(* Logix 5000 project; controller TestController vendor 1 type 14 code 166 rev 32.11; software revision 32.02 *)
// This is a test project

TASK Continuous (continuous, watchdog 500 ms) : MainProgram   // Test continuous task
TASK Event (event, rate 11 ms, priority 10, watchdog 500 ms) : EventProgram   // TestEvent Task
TASK Periodic (periodic, rate 10 ms, priority 10, watchdog 500 ms) : EPProgram, NProgram, Empty

MODULES
   Local : vendor 1 type 14 code 166 (ICP 0, rev 32.11)
      Local_Mod_4 : 1756sc-CTR8 (ICP 4, rev 1.1, Output RPI 10 ms)
      Local_Mod_6 : 1756-CNB (ICP 6, rev 11.1)
         LM6C1 : 1407-CGCM (ControlNet 2, rev 4.1, Output RPI 5 ms)
      Local_Mod_8 : vendor 1 type 14 code 166 (ICP 8, rev 32.1, $6765098e$ RPI 20 ms)
      NetworkController : vendor 1 type 14 code 166 (Ethernet 192.168.1.232, rev 32.1)
      Local_Mod_5 : 1756-M02AE (ICP 5, rev 32.1, MotionEvent RPI 1000 ms, MotionAsync RPI 25 ms)
      TestEtap : 1783-ETAP (Ethernet 192.168.1.247, rev 2.1)
      Local_Mod_1 : 1756-EN2T (ICP 1, Ethernet 1.1.1.1, rev 11.1)
         L1M1 : 1756-EN2T (Ethernet 2.2.2.2, rev 11.1, Output RPI 10 ms)
            L1M1D1 : 1756-IT6I (ICP 1, rev 1.1, Input RPI 100 ms)
         L1M3 : 1732E-IB16M12DR (Ethernet 54.3.56.6, rev 1.1, Input RPI 20 ms)
         L1M2 : 1734-AENT (Ethernet 3.3.3.3, rev 5.1, Output RPI 20 ms)
            L1M2D1 : 1734-IV8 (PointIO 1, rev 3.1)
      RackIO : 1756-EN2T (Ethernet 10.10.10.10, rev 11.1, Output RPI 10 ms)   // This is a test EN2T module
         Rack_Mod_1 : 1756-IB16 (ICP 1, rev 3.1)
         Rack_Mode_3 : 1756-IB16 (ICP 3, rev 3.1)
              RackIO:3:I.Data.0   // IO Description
         Rack_Mod_2 : 1756-IF8 (ICP 2, rev 1.1, Input RPI 100 ms)   // Ths is a test IF8
      TestCard : 1756-EN2T (Ethernet Host-Name.Com1234d5asdvdlkjadvasdfasdfasddfasdfasdfasdasdfasdfda, rev 11.1)   // This is a test EN2T module
      ImportTest : 1756-EN2T (ICP 7, Ethernet 10.2.10.4, rev 11.1)   // This is a test EN2T module
      FlexBus : 1794-AENT (Ethernet 192.168.1.251, rev 4.1, Output RPI 20 ms)
         FB1 : 1794-IB16 (Flex 0, rev 1.1)
         FB2 : 1794-IB16 (Flex 1, rev 1.1)
      Local_Mod_9 : 1756-DHRIO (ICP 9, rev 7.1, Input RPI 25 ms)
         RIOChA1 : 1747-ASB (RIO 1, rev 1.1, Output RPI 48 ms)
         RIOChA2 : 1794-ASB (RIO 2, rev 1.1, Output RPI 48 ms)
         RIOChB1 : 1771-ASB (RIO 0, rev 1.1, Output RPI 48 ms)
      Local_Mod_3 : 1756-RIO (ICP 3, rev 3.1, Output RPI 20 ms)
      Local_Mod_2 : MVI56E-MCM (ICP 2, rev 3.1, Output RPI 5 ms)
      FlexIO : 5094-AEN2TR (Ethernet 10.11.12.13, rev 4.1)
         Flex_Mod_1 : 5094-IF8 (5094 1, rev 2.1, StandardDataDriven RPI 100 ms)
         Flex_Mod_2 : 5094-OB16 (5094 2, rev 2.1, StandardDataDriven RPI 5 ms)
         Flex_Mod_3 : 5094-IB16 (5094 3, rev 2.1, StandardDataDriven RPI 5 ms)
         Flex_Mod_4 : 5094-IB32 (5094 4, rev 2.1, StandardDataDriven RPI 5 ms)
         Flex_Mod_5 : 5094-OF8 (5094 5, rev 2.1, StandardDataDriven RPI 100 ms)
         Flex_Mod_6 : 5094-IY8 (5094 6, rev 3.1, StandardDataDriven RPI 100 ms)
         Flex_Mod_7 : 5094-HSC (5094 7, rev 2.1, StandardDataDriven RPI 80 ms)
END_MODULES

TYPE AlarmType :   // This is a test alarm type
STRUCT
   DigitalMember : CAM;   // Test digital member
END_STRUCT
END_TYPE

TYPE BoolTest :   // This is a test
STRUCT
   Member01 : BOOL;
   Member02 : BOOL;
   Member04 : BOOL;
   Member05 : BOOL;
END_STRUCT
END_TYPE

TYPE FakeString :   // This is a type
STRUCT
   LEN : DINT;
   DATA : SINT[23];
END_STRUCT
END_TYPE

TYPE ModuleType :   // This is a test of a type that references Module-Defined types
STRUCT
   AIChannel : CHANNEL_AI:O:0;   // This is a test
   TestChannel : CHANNEL_AI:O:0;   // This is a test
END_STRUCT
END_TYPE

TYPE MyStringType :   // This is a test string type
STRUCT
   LEN : DINT;
   DATA : SINT[100];
END_STRUCT
END_TYPE

TYPE TestType :   // this is a test
STRUCT
   Timers : TIMER[5];
   Number : DINT;
   Flag : BOOL;
END_STRUCT
END_TYPE

ADD_ON_INSTRUCTION aoi_Test   (* revision 1.2 *)
// Help:
// This is a test aoi definitio that was built for purposes of exporting data to examine the structure of the L5X
VAR_INPUT
   InputTest : BOOL; {visible}
   OutputTest : DINT; {access Read Only, visible}
END_VAR
VAR_IN_OUT
   InOutTest : SimpleType; {required}
END_VAR
VAR_INPUT
   Config : INT; {access None, required}
   Test : BOOL; {access None}
END_VAR
VAR_IN_OUT
   InOutArray : REAL[5]; {required}
END_VAR
VAR_INPUT
   New : DINT; {required}
   Alias : ALIAS FOR LocalBool; {access None}   // This is an alias
END_VAR
VAR
   LocalBool : BOOL; {access None}
   LocalComplex : SimpleType;   // Description Test
   LocalArray : DINT[5]; {access None}
   LocalString : STRING; {access None}
END_VAR

ROUTINE Logic   (* ladder *)
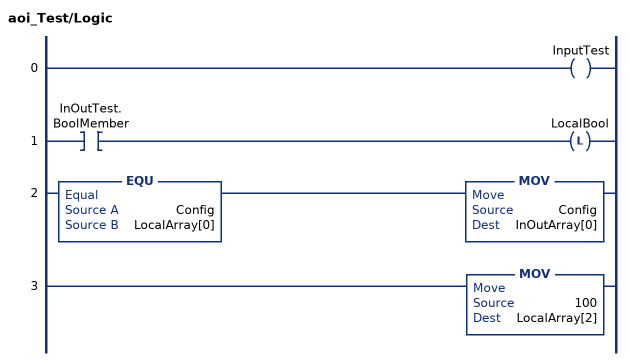
   0: OTE(InputTest);
   1: XIC(InOutTest.BoolMember)OTL(LocalBool);
   2: EQU(Config,LocalArray[0])MOV(Config,InOutArray[0]);
   3: MOV(100,LocalArray[2]);
END_ROUTINE

ROUTINE Prescan   (* ladder *)
END_ROUTINE
END_ADD_ON_INSTRUCTION

VAR_GLOBAL   (* controller tags *)
   _Test : DINT;
   AliasTag : ALIAS FOR Another;
   Another : DINT := 4;
   aoiTestInstance : aoi_Test;
   AsciiTag : SINT := '$10';
   Consumer : DINT;
   DateTimeNs : LINT := 1641016800100100100;
   EPProgram : PHASE;
   FakeStringTag : FakeString;
   MultiDimensionalArray : DINT[3,5];
   NewTag : ComplexType; {access None}
   ProducedTag : DINT; {produced}
   ProviderTag : TIMER; {produced}
   RealArray : REAL[5];
   SimpleArray : DINT[10]; {access Read Only}   // This is a test
   SimpleBool : BOOL;   // A simple boolean tag element
   SimpleDint : DINT := 123392; {access None}
   SimpleInt : INT := 4321; {access None}   // This is a simple integer tag
   SimpleLint : LINT := 123; {access None}
   SimpleReal : REAL := 1.23; {access None}
   SimpleSint : SINT := 16#0c; {access None}
        .0   // This is a test
   SimpleString : STRING := 'This is a test string type';   // This is a test string
   SimpleUDint : UDINT;
   SimpleUInt : UINT;
   SimpleULint : ULINT;
   SimpleUSint : USINT := 255;
   SintArray : SINT[100] := ([0] := '$01', [1] := '$02', [2] := '$03', [3] := '$04', [4] := '$05', [5] := '$06', [6] := '$07', [7] := '$08', [8] := '$09', [9] := '$0A', [10] := '$0B', [11] := '$0C', [12] := '$0D', [13] := '$0E', [14] := '$0F', [15] := '$10', [16] := '$11', [17] := '$12', [18] := '$13', [19] := '$14', [20] := '$15', [21] := '$16', [22] := '$17', [23] := '$18', [24] := '$19', [25] := '$1A', [26] := '$1B', [27] := '$1C', [28] := '$1D', [29] := '$1E', [30] := '$1F', [31] := ' ', [32] := '!', [33] := '"', [34] := '#', [35] := '$$', [36] := '%', [37] := '&', [38] := '$'', [39] := '(', [40] := ')', [41] := '*', [42] := '+', [43] := ',', [44] := '-', [45] := '.', [46] := '/', [47] := '0', [48] := '1', [49] := '2', [50] := '3', [51] := '4', [52] := '5', [53] := '6', [54] := '7', [55] := '8', [56] := '9', [57] := ':', [58] := ';', [59] := '<',
        [60] := '=', [61] := '>', [62] := '?', [63] := '@', [64] := 'A', [65] := '$FF');
   StringArray : STRING[5];   // String Array
   TagParameter : SimpleType; {access None}
   TestAlarmTag : ALARM; {access None}   // Alarm
   TestAlarmType : AlarmType;
   TestAnalogAlarm : ALARM_ANALOG;
   TestArray : DINT[1,1,2];
   TestArrayOfArray : ArrayType[5];   // tessting an array of arrays
   TestArrayTag : ArrayType := (LintArray[0] := 1645509600000000); {access Read Only}   // Base
   TestComplexTag : ComplexType := (SimpleMember.LintMember := 2); {access None}   // Base
   TestDigitalAlarm : ALARM_DIGITAL;
   TestSimpleTag : SimpleType := (IntMember := 14, DintMember := '$00$00$00$01'); {access Read Only}   // This is a test tag with a description or comment.
   TestStringTag : MyStringType := 'This is a $$ tests'; {access None}   // String
        .DATA   // Data
   TestTimer : TIMER := (PRE := 1000); {access None}
        .PRE   // Test Timer PRE
   TimerArray : TIMER[5] := ([0].PRE := 5000);   // Base Timer
        [1]   // Index 1
        [1].PRE   // PRE 1
   XIC : BOOL;
END_VAR

PROGRAM Empty
END_PROGRAM

PROGRAM EPProgram
// Test Equipment Phase Program
END_PROGRAM

PROGRAM EventProgram   (* main routine Main *)

ROUTINE Main   (* ladder *)
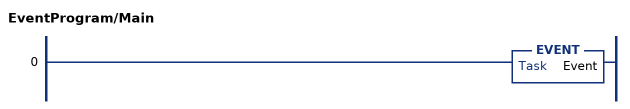
   0: EVENT(Event);
END_ROUTINE
END_PROGRAM

PROGRAM FolderProgram
END_PROGRAM

PROGRAM MainProgram   (* main routine Main *)
VAR
   Action_000 : SFC_ACTION := (Status := 16#0020_0000, PauseTimer := 1);
   ADD_01 : FBD_MATH;
   BufferTag : BOOL;
   Channel : DINT;
   connection : DINT; {access None}
   InputParameter : DINT;
   LPF_01 : FILTER_LOW_PASS := (Order := 1, RTSTime := 1);
   OutputParameter : DINT;
   Step_000 : SFC_STEP := (Status := 16#0020_0000, PauseTimer := 1);
   Step_001 : SFC_STEP := (Status := 16#0020_0000, PauseTimer := 1);
   Step_002 : SFC_STEP := (Status := 16#0020_0000, PauseTimer := 1);
   Step_003 : SFC_STEP := (Status := 16#0020_0000, PauseTimer := 1);
   Step_004 : SFC_STEP := (Status := 16#0020_0000, PauseTimer := 1);
   Stop_000 : SFC_STOP;
   Test : SERIAL_PORT_CONTROL := (POS := 12);
   TestSimpleTag : SimpleType;
   Tran_000 : BOOL;
   Tran_001 : BOOL;
   Tran_002 : BOOL;
END_VAR

ROUTINE FBD   (* function block diagram *)
   SHEET 1
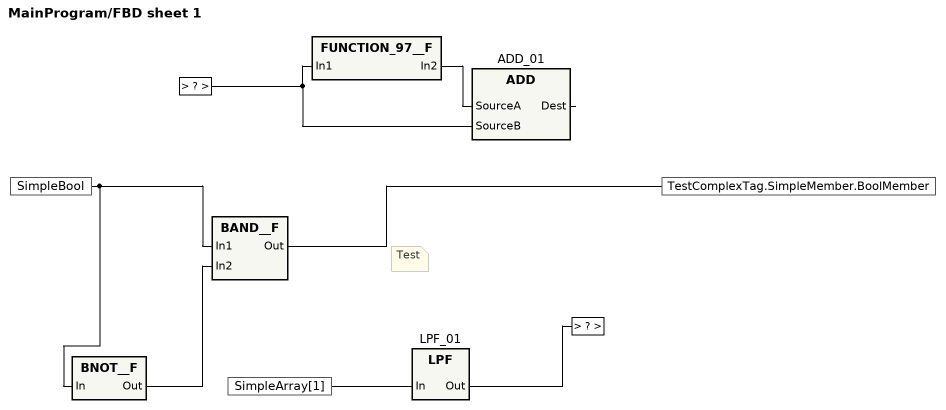
   // Test
   BNOT__F_1 : BNOT__F(In := SimpleBool);
   BAND__F_2 : BAND__F(In1 := SimpleBool, In2 := BNOT__F_1.Out);
   LPF_01 : LPF(In := SimpleArray[1]);
   WIRE(?) := LPF_01.Out;
   FUNCTION_97__F_3 : FUNCTION_97__F(In1 := WIRE(?));
   ADD_01 : ADD(SourceA := FUNCTION_97__F_3.In2, SourceB := WIRE(?));   // unwired pins: Dest
   TestComplexTag.SimpleMember.BoolMember := BAND__F_2.Out;
END_ROUTINE

ROUTINE Main   (* ladder *)
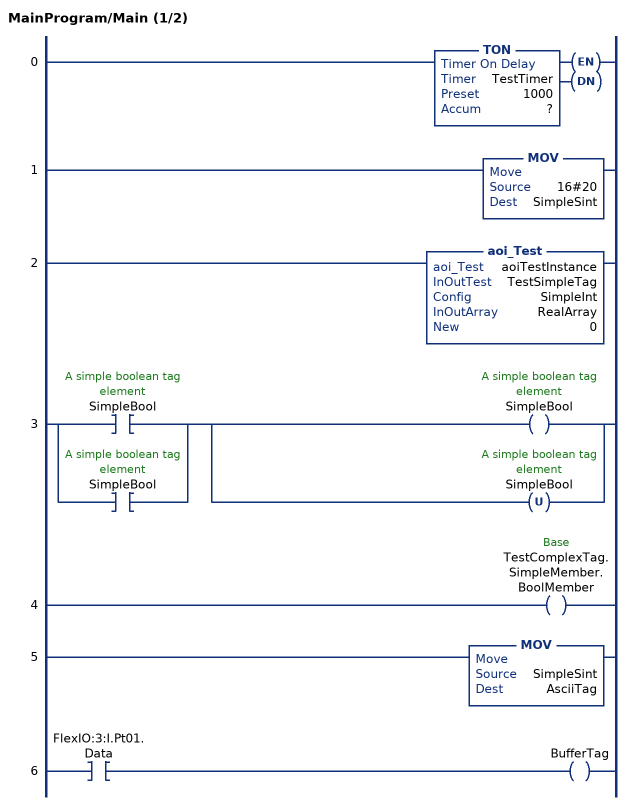
   0: TON(TestTimer,?,?);
   1: MOV(16#20,SimpleSint);
   2: aoi_Test(aoiTestInstance,TestSimpleTag,SimpleInt,RealArray,0);
   3: [XIC(SimpleBool) ,XIC(SimpleBool) ][OTE(SimpleBool) ,OTU(SimpleBool) ];
   4: OTE(TestComplexTag.SimpleMember.BoolMember);
   5: MOV(SimpleSint,AsciiTag);
   6: XIC(FlexIO:3:I.Pt01.Data)OTE(BufferTag);
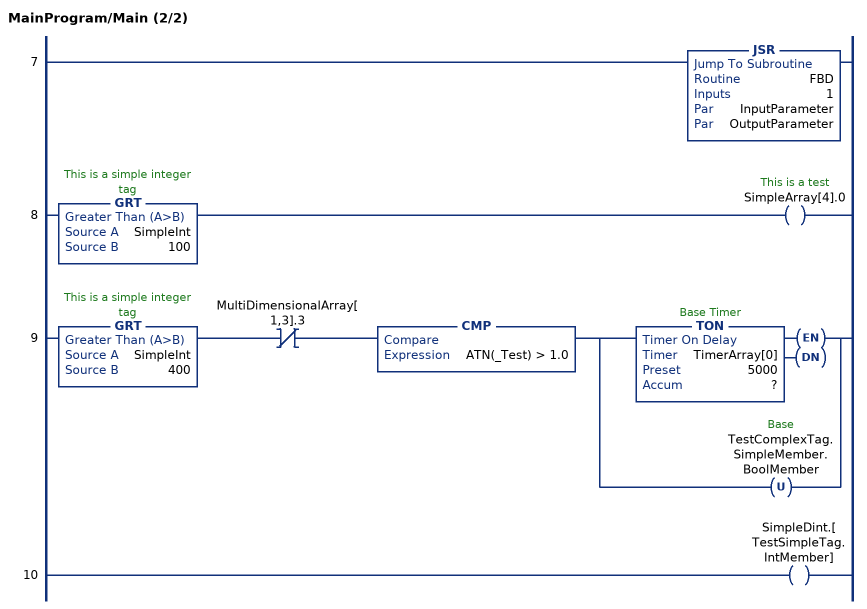
   7: JSR(FBD,1,InputParameter,OutputParameter);
   8: GRT(SimpleInt,100)OTE(SimpleArray[4].0);
   9: GRT(SimpleInt,400)XIO(MultiDimensionalArray[1,3].3)CMP(ATN(_Test) > 1.0)[TON(TimerArray[0],?,?) ,OTU(TestComplexTag.SimpleMember.BoolMember) ];
   10: OTE(SimpleDint.[TestSimpleTag.IntMember]);
END_ROUTINE

ROUTINE SFC   (* sequential function chart *)
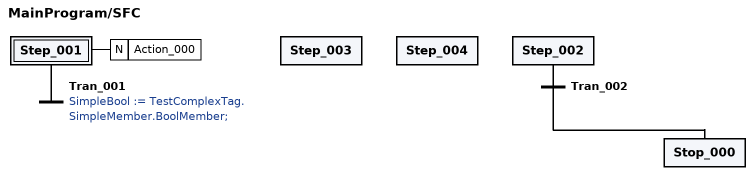
   INITIAL_STEP Step_001:
      ACTION Action_000 (N):
         
      END_ACTION
   END_STEP
   STEP Step_002:
   END_STEP
   TRANSITION Tran_001 FROM Step_001 TO ()
      := SimpleBool := TestComplexTag.SimpleMember.BoolMember;
   END_TRANSITION
   TRANSITION Tran_002 FROM Step_002 TO Stop_000
      := 
   END_TRANSITION
   STEP Step_003:
   END_STEP
   STEP Step_004:
   END_STEP
   STOP Stop_000;
END_ROUTINE

ROUTINE ST   (* structured text *)
   SimpleBool := TestComplexTag.SimpleMember.BoolMember;
   
   _Test := 100 + ABS((TestSimpleTag.IntMember+14)/2);
   
   _Test := TestSimpleTag.DintMember MOD 100;
   
   
   
END_ROUTINE
END_PROGRAM

PROGRAM NProgram   (* main routine Main, fault routine Fault *)
// Test Program
VAR_IN_OUT
   InOutTag : INT;
END_VAR
VAR_INPUT
   InTag : DINT;
END_VAR
VAR
   LocalBool : BOOL;
   LocalComplex : ComplexType;
   LocalDint : DINT := 1234;
   LocalReal : REAL;
   LocalSimlpe : SimpleType;
END_VAR
VAR_OUTPUT
   OutTag : DINT;
END_VAR
VAR {public}
   PublicInt : INT;
END_VAR

ROUTINE Fault   (* ladder *)
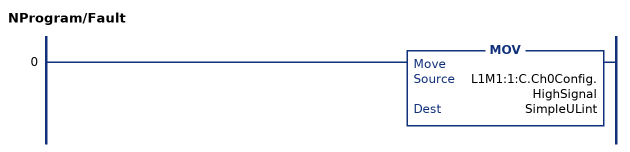
   0: MOV(L1M1:1:C.Ch0Config.HighSignal,SimpleULint);
END_ROUTINE

ROUTINE Main   (* ladder *)
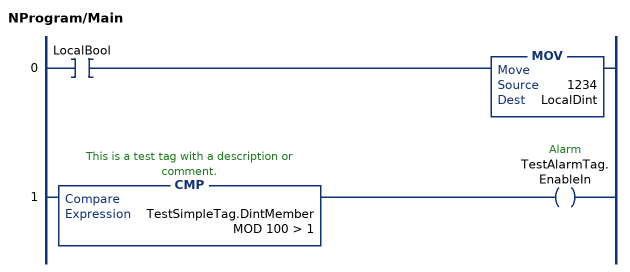
   0: XIC(LocalBool)MOV(1234,LocalDint);
   1: CMP(TestSimpleTag.DintMember MOD 100 > 1)OTE(TestAlarmTag.EnableIn);
END_ROUTINE
END_PROGRAM
